PROGRAM MAIN
VAR
END_VAR

END_PROGRAM

(* stored: Version 1.1.0.1, ProductVersion 3.1.4024.11
   POU MAIN: Id {3c8728e6-ac66-400a-b515-5b76be139338}, SpecialFunc None *)
